// TIA Portal project "Progetto4" (V15.1)

(* hardware
DEVICE "S7-1200 station_2"  S7-1200 Station
   slot 0: "Telaio di montaggio_0"  S7-1200 Rack  Rack  V1.0
   slot 1: "IO-Device"  CPU 1214C DC/DC/DC  6ES7 214-1AG40-0XB0  V4.2
DEVICE "S7-1200 station_1"  S7-1200 Station
   slot 0: "Telaio di montaggio_0"  S7-1200 Rack  Rack  V1.0
   slot 1: "IO-Controller"  CPU 1214C DC/DC/DC  6ES7 214-1AG40-0XB0  V4.2
*)

// ===== PLC "IO-Controller"  CPU 1214C DC/DC/DC =====

VAR_GLOBAL   // PLC tag table "Tabella delle variabili standard"
   "Connetti" AT %I0.0 : Bool;
   "Disconnetti" AT %I0.1 : Bool;
END_VAR

DATA_BLOCK "DatiTx"   // DB2
{ S7_Optimized_Access := 'FALSE' }
VERSION : 0.1
   VAR
      TestBool : Bool;
      TestInt : Int;
   END_VAR
BEGIN
END_DATA_BLOCK

DATA_BLOCK "DatiRx"   // DB3
{ S7_Optimized_Access := 'FALSE' }
VERSION : 0.1
   VAR
      TestBool : Bool;
      TestInt : Int;
   END_VAR
BEGIN
END_DATA_BLOCK

// folder: System blocks/Program resources

DATA_BLOCK "IO-Controller_Connection_DB"   // DB4
{ S7_Optimized_Access := 'TRUE' }
AUTHOR : SIMATIC
FAMILY : MC7Plus
NAME : TC_IP_v4
VERSION : 1.0
// stored: InstanceOfName TCON_IP_v4
"TCON_IP_v4"
BEGIN
   ID := 1;
   InterfaceId := 64;
   RemotePort := 2000;
   ActiveEstablished := true;
   RemoteAddress.ADDR[1] := 192;
   RemoteAddress.ADDR[2] := 168;
   RemoteAddress.ADDR[4] := 2;
END_DATA_BLOCK

// folder: (top level)

ORGANIZATION_BLOCK "Main"   // OB1, LAD, ProgramCycle
TITLE = "Main Program Sweep (Cycle)"
{ S7_Optimized_Access := 'TRUE' }
VERSION : 0.1
   VAR_INPUT
      Initial_Call : Bool;   // Initial call of this OB
      Remanence : Bool;   // =True, if remanent data are available
   END_VAR
BEGIN

REGION Network 1
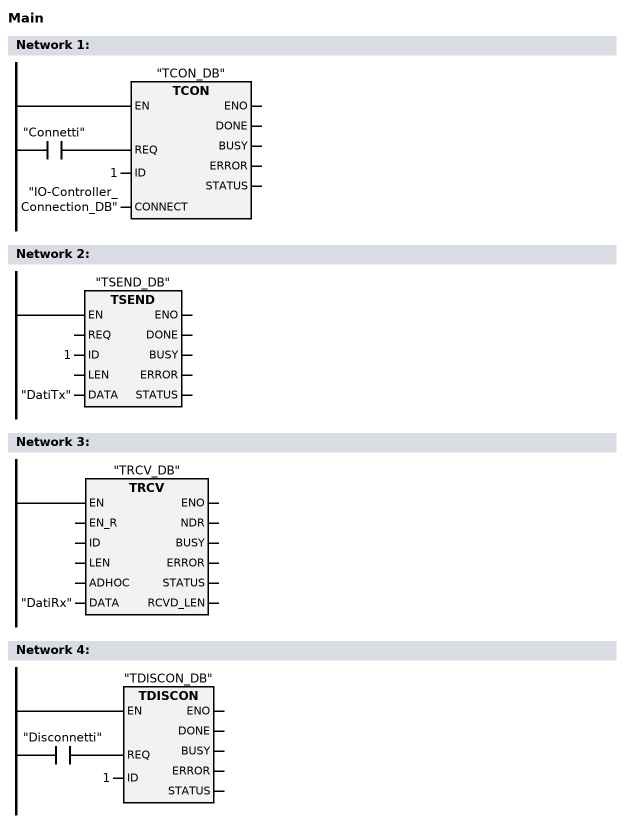
   "TCON_DB"(REQ := "Connetti", ID := 1, CONNECT := "IO-Controller_Connection_DB");   // TCON
END_REGION

REGION Network 2
   "TSEND_DB"(ID := 1, DATA := "DatiTx");   // TSEND
END_REGION

REGION Network 3
   "TRCV_DB"(DATA := "DatiRx");   // TRCV
END_REGION

REGION Network 4
   "TDISCON_DB"(REQ := "Disconnetti", ID := 1);   // TDISCON
END_REGION
END_ORGANIZATION_BLOCK

// ===== PLC "IO-Device"  CPU 1214C DC/DC/DC =====

DATA_BLOCK "DatiRx"   // DB5
{ S7_Optimized_Access := 'FALSE' }
VERSION : 0.1
   VAR
      testBool : Bool;
      testInt : Int;
   END_VAR
BEGIN
END_DATA_BLOCK

DATA_BLOCK "DatiTx"   // DB6
{ S7_Optimized_Access := 'FALSE' }
VERSION : 0.1
   VAR
      testBool : Bool;
      testInt : Int;
   END_VAR
BEGIN
END_DATA_BLOCK

// folder: System blocks/Program resources

DATA_BLOCK "IO-Device_Connection_DB"   // DB1
{ S7_Optimized_Access := 'TRUE' }
AUTHOR : SIMATIC
FAMILY : MC7Plus
NAME : TC_IP_v4
VERSION : 1.0
// stored: InstanceOfName TCON_IP_v4
"TCON_IP_v4"
BEGIN
   ID := 1;
   InterfaceId := 64;
   LocalPort := 2000;
   RemoteAddress.ADDR[1] := 192;
   RemoteAddress.ADDR[2] := 168;
   RemoteAddress.ADDR[4] := 1;
END_DATA_BLOCK

// folder: (top level)

ORGANIZATION_BLOCK "Main"   // OB1, LAD, ProgramCycle
TITLE = "Main Program Sweep (Cycle)"
{ S7_Optimized_Access := 'TRUE' }
VERSION : 0.1
   VAR_INPUT
      Initial_Call : Bool;   // Initial call of this OB
      Remanence : Bool;   // =True, if remanent data are available
   END_VAR
BEGIN

REGION Network 1
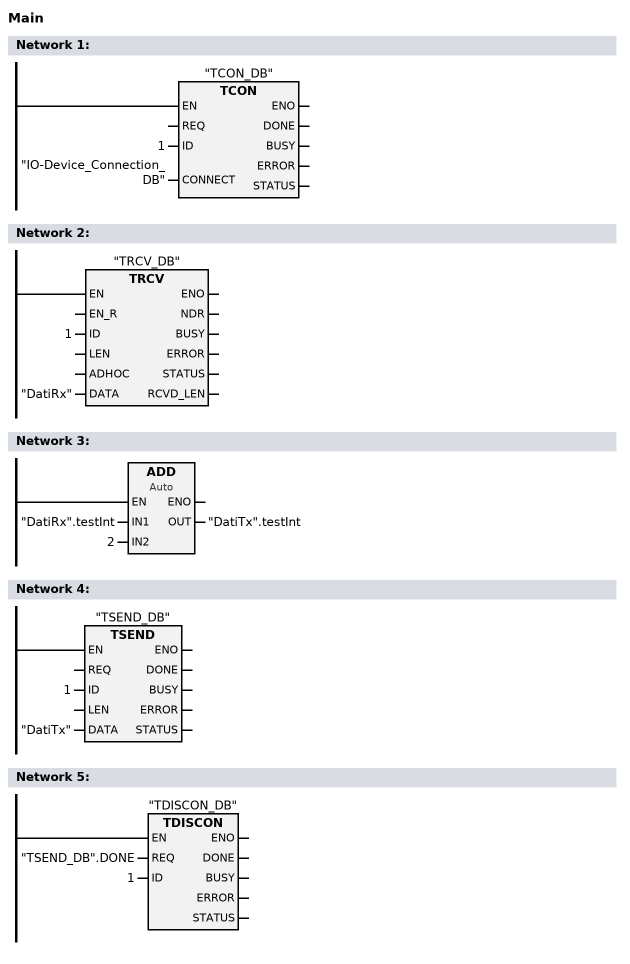
   "TCON_DB"(ID := 1, CONNECT := "IO-Device_Connection_DB");   // TCON
END_REGION

REGION Network 2
   "TRCV_DB"(ID := 1, DATA := "DatiRx");   // TRCV
END_REGION

REGION Network 3
   RUNG wire#powerrail
      Add(in1 := "DatiRx".testInt, in2 := 2, out => "DatiTx".testInt)
   END_RUNG
   // the same network as SCL:
   "DatiTx".testInt := "DatiRx".testInt + 2;
END_REGION

REGION Network 4
   "TSEND_DB"(ID := 1, DATA := "DatiTx");   // TSEND
END_REGION

REGION Network 5
   "TDISCON_DB"(REQ := "TSEND_DB".DONE, ID := 1);   // TDISCON
END_REGION
END_ORGANIZATION_BLOCK